(* CoDeSys 2.3 export: FB_STATION_7.EXP *)

(* POU fb_station_7, FBD *)
FUNCTION_BLOCK fb_station_7
VAR_INPUT
	blinkTakt							:	BOOL;
	notaus								:	BOOL;
	startTaster							:	BOOL;
	sensor_rotaryStep				:	BOOL;
	sensor_partStartPos				:	BOOL;
	sensor_partEndPos				:	BOOL;
	sensor_punchProximity			:	BOOL;
	sensor_punchFullyExtended		:	BOOL;
	sensor_drillProximity				:	BOOL;
	sensor_drillUpperLimit			:	BOOL;
	sensor_drillLowerLimit			:	BOOL;
	handshake_start					:	BOOL;
	handshake_nextBusy				:	BOOL;
END_VAR
VAR_OUTPUT
	aktor_rotaryMotor					:	BOOL;
	aktor_punch						:	BOOL;
	aktor_lowerDrill					:	BOOL;
	aktor_raiseDrill					:	BOOL;
	aktor_drill							:	BOOL;
	aktor_drillPunch					:	BOOL;
	aktor_emergencyIndicator		:	BOOL;
	aktor_initPosIndicator				:	BOOL;
	aktor_pbStartIndicator			:	BOOL;
	aktor_lampState0					:	BOOL;
	aktor_lampState1					:	BOOL;
	aktor_lampState2					:	BOOL;
	aktor_lampState3					:	BOOL;
	aktor_lampState4					:	BOOL;
	aktor_lampState5					:	BOOL;
	aktor_lampState6					:	BOOL;
	aktor_lampState7					:	BOOL;
	aktor_lampState8					:	BOOL;
	handshake_busy					:	BOOL;
	handshake_startNext				:	BOOL;
END_VAR
VAR
	sr_emergencyHalt	:	SR;
	calcTransitions		:	CALC_TRANSITIONS;
	seqCtrl				:	SEQUENTIAL_CTRL;
	actuatorCtrl			:	ACTUATOR_CTRL;
	calcFlags				:	CALC_FLAGS;
	indicatorCtrl			:	INDICATOR_CTRL;
END_VAR
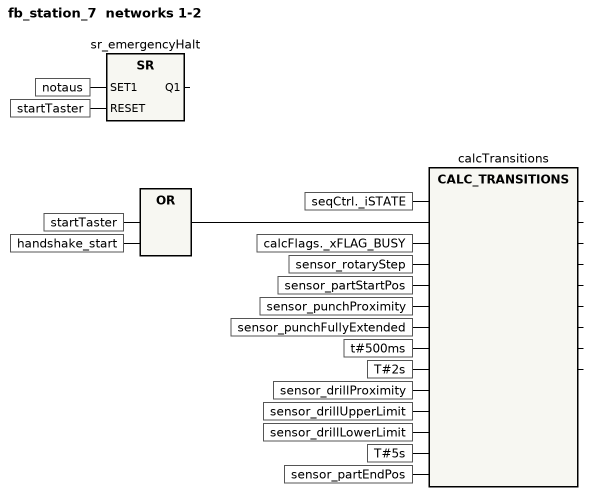
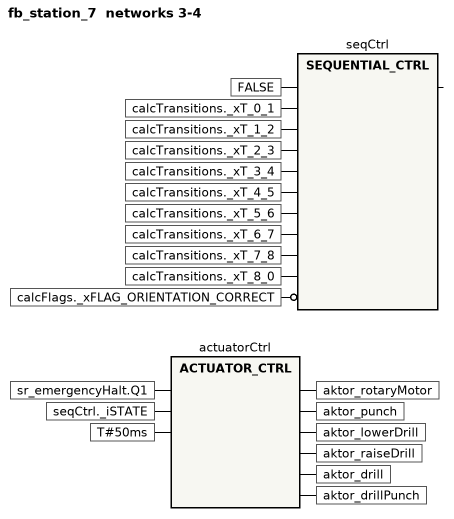
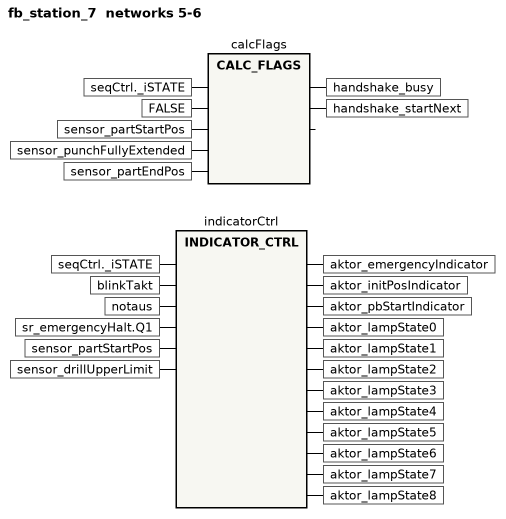
_FBD_ (* Function Block Diagram *)
NETWORK 1 emergencyHalt: (* Sets when Emergency is active, resets if it's not and the start button is pressed. *)
	sr_emergencyHalt:SR(SET1: notaus, RESET: startTaster)
NETWORK 2 transitions: (* Gets sensor values and calculates transitional conditions. *)
	calcTransitions:CALC_TRANSITIONS(seqCtrl._iSTATE, OR(startTaster, handshake_start), calcFlags._xFLAG_BUSY, sensor_rotaryStep, sensor_partStartPos, sensor_punchProximity, sensor_punchFullyExtended, t#500ms, T#2s, sensor_drillProximity, sensor_drillUpperLimit, sensor_drillLowerLimit, T#5s, sensor_partEndPos)
NETWORK 3 stateMachine: (* Saves and outputs the current machine state, increments if the corresponding transitional condition is met, returning back to state 0 from state 8. If the jump flag is set, steps 5,6 and 7 are skipped. *)
	seqCtrl:SEQUENTIAL_CTRL(FALSE, calcTransitions._xT_0_1, calcTransitions._xT_1_2, calcTransitions._xT_2_3, calcTransitions._xT_3_4, calcTransitions._xT_4_5, calcTransitions._xT_5_6, calcTransitions._xT_6_7, calcTransitions._xT_7_8, calcTransitions._xT_8_0, NOT calcFlags._xFLAG_ORIENTATION_CORRECT)
NETWORK 4 actuators: (* Controls which actuators are active in each state, all actuators get turned off in case of an emergency. *)
	actuatorCtrl:ACTUATOR_CTRL(sr_emergencyHalt.Q1, seqCtrl._iSTATE, T#50ms, out 2 => aktor_punch, out 3 => aktor_lowerDrill, out 4 => aktor_raiseDrill, out 5 => aktor_drill, out 6 => aktor_drillPunch) => aktor_rotaryMotor
NETWORK 5 flags: (* Sets various flags for communication with other stations and between POUs of this station. *)
	calcFlags:CALC_FLAGS(seqCtrl._iSTATE, FALSE, sensor_partStartPos, sensor_punchFullyExtended, sensor_partEndPos, out 2 => handshake_startNext) => handshake_busy
NETWORK 6 stateIndicator: (* Controls Indicator lights. *)
	indicatorCtrl:INDICATOR_CTRL(seqCtrl._iSTATE, blinkTakt, notaus, sr_emergencyHalt.Q1, sensor_partStartPos, sensor_drillUpperLimit, out 2 => aktor_initPosIndicator, out 3 => aktor_pbStartIndicator, out 4 => aktor_lampState0, out 5 => aktor_lampState1, out 6 => aktor_lampState2, out 7 => aktor_lampState3, out 8 => aktor_lampState4, out 9 => aktor_lampState5, out 10 => aktor_lampState6, out 11 => aktor_lampState7, out 12 => aktor_lampState8) => aktor_emergencyIndicator
_END_FBD_
(* the same logic as Structured Text *)
(* Network 1 *)
sr_emergencyHalt(SET1 := notaus, RESET := startTaster);
(* Network 2 *)
calcTransitions(seqCtrl._iSTATE, startTaster OR handshake_start, calcFlags._xFLAG_BUSY, sensor_rotaryStep, sensor_partStartPos, sensor_punchProximity, sensor_punchFullyExtended, t#500ms, T#2s, sensor_drillProximity, sensor_drillUpperLimit, sensor_drillLowerLimit, T#5s, sensor_partEndPos);
(* Network 3 *)
seqCtrl(FALSE, calcTransitions._xT_0_1, calcTransitions._xT_1_2, calcTransitions._xT_2_3, calcTransitions._xT_3_4, calcTransitions._xT_4_5, calcTransitions._xT_5_6, calcTransitions._xT_6_7, calcTransitions._xT_7_8, calcTransitions._xT_8_0, NOT calcFlags._xFLAG_ORIENTATION_CORRECT);
(* Network 4: see the listing above *)
(* Network 5: see the listing above *)
(* Network 6: see the listing above *)
END_FUNCTION_BLOCK
